TYPE Box :
STRUCT
  BoxId : INT;
  DetectedAt : LWORD;
  CompletionRatio : LREAL;
END_STRUCT
END_TYPE

(* stored: Version 1.1.0.1
   DUT Box: Id {ea428213-be68-4453-a3d6-0330e86964c3} *)
